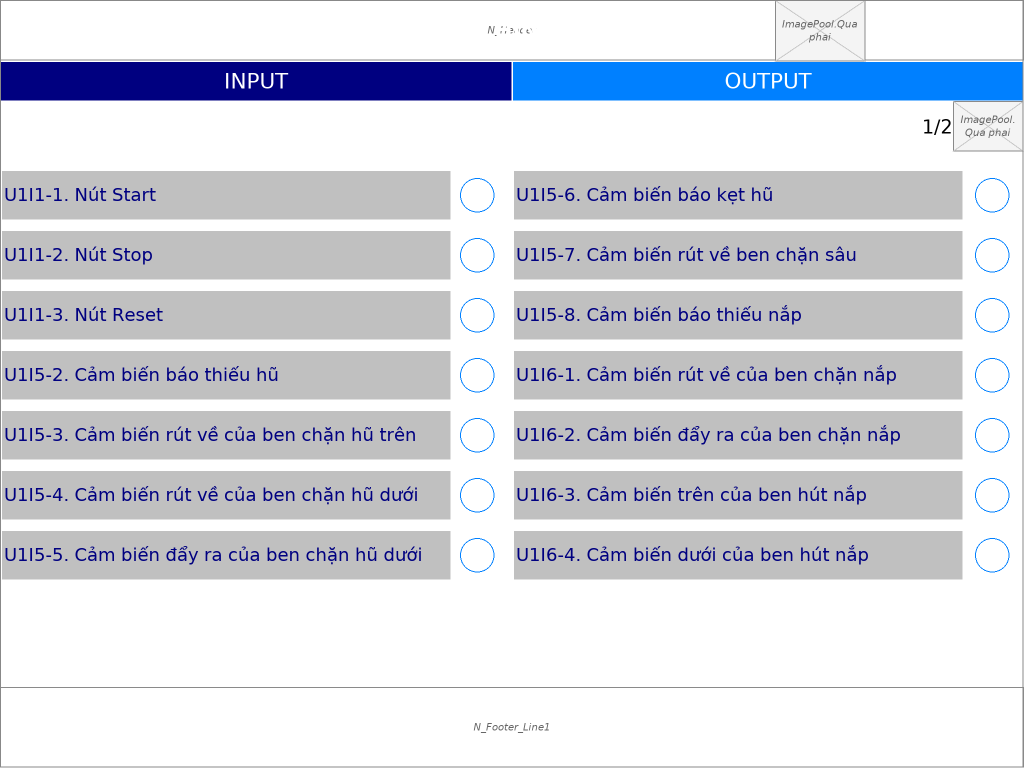
VISUALIZATION N_PLC_I1  // 1024x768
    Frame (0,687 1024x80)
        shows N_Footer_Line1()
    Frame (0,0 1024x60)
        shows N_Header()
    Textfield (353,5 400x50), "MÀN HÌNH IO LINE 1"
    Rectangle (0,61 512x40), "INPUT"
        OnMouseClick: change screen: N_PLC_I1
    Rectangle (512,61 512x40), "OUTPUT"
        OnMouseClick: change screen: N_PLC_O1
    Image (775,0 90x61), image: ImagePool.Qua phai
        OnMouseClick: change screen: N_PLC_I2
    Rectangle (1,350 450x50), "U1I5-2. Cảm biến báo thiếu hũ"
    Rectangle (1,410 450x50), "U1I5-3. Cảm biến rút về của ben chặn hũ trên"
    Rectangle (1,470 450x50), "U1I5-4. Cảm biến rút về của ben chặn hũ dưới"
    Rectangle (1,530 450x50), "U1I5-5. Cảm biến đẩy ra của ben chặn hũ dưới"
    Rectangle (1,170 450x50), "U1I1-1. Nút Start"
    Rectangle (1,230 450x50), "U1I1-2. Nút Stop"
    Rectangle (1,290 450x50), "U1I1-3. Nút Reset"
    Ellipse (460,178 34x34), colour toggle: GVL_IO.bStart, input disabled if: true
    Ellipse (460,238 34x34), colour toggle: GVL_IO.bStop, input disabled if: true
    Ellipse (460,298 34x34), colour toggle: GVL_IO.bReset, input disabled if: true
    Ellipse (460,358 34x34), colour toggle: PR_Line01.fb_CupSupply.bCupEmpty, input disabled if: true
    Ellipse (460,418 34x34), colour toggle: PR_Line01.fb_CupSupply.fbCylinder_Up.bAtRetract, input disabled if: true
    Ellipse (460,478 34x34), colour toggle: PR_Line01.fb_CupSupply.fbCylinder_Dw.bAtRetract, input disabled if: true
    Ellipse (460,538 34x34), colour toggle: PR_Line01.fb_CupSupply.fbCylinder_Dw.bAtExtend, input disabled if: true
    Rectangle (513,530 450x50), "U1I6-4. Cảm biến dưới của ben hút nắp"
    Rectangle (513,170 450x50), "U1I5-6. Cảm biến báo kẹt hũ"
    Rectangle (513,230 450x50), "U1I5-7. Cảm biến rút về ben chặn sâu"
    Rectangle (513,290 450x50), "U1I5-8. Cảm biến báo thiếu nắp"
    Rectangle (513,350 450x50), "U1I6-1. Cảm biến rút về của ben chặn nắp"
    Rectangle (513,410 450x50), "U1I6-2. Cảm biến đẩy ra của ben chặn nắp"
    Rectangle (513,470 450x50), "U1I6-3. Cảm biến trên của ben hút nắp"
    Ellipse (975,178 34x34), colour toggle: PR_Line01.fb_CupSupply.bCupDrop, input disabled if: true
    Ellipse (975,538 34x34), colour toggle: PR_Line01.fb_LidSupply.fbCylinder_Suction.bAtExtend, input disabled if: true
        toggle GVL_OF_VU.bSensorOutOfLid[2]
    Ellipse (975,238 34x34), colour toggle: PR_Line01.fb_WormWeight.fbCylinder.bAtRetract, input disabled if: true
    Ellipse (975,298 34x34), colour toggle: PR_Line01.fb_LidSupply.bLidEmpty, input disabled if: true
    Ellipse (975,358 34x34), colour toggle: PR_Line01.fb_LidSupply.fbCylinder_LidStopper.bAtRetract, input disabled if: true
    Ellipse (975,418 34x34), colour toggle: PR_Line01.fb_LidSupply.fbCylinder_LidStopper.bAtExtend, input disabled if: true
    Ellipse (975,478 34x34), colour toggle: PR_Line01.fb_LidSupply.fbCylinder_Suction.bAtRetract, input disabled if: true
    Rectangle (886,102 103x50), "1/2"
    Image (953,101 70x50), image: ImagePool.Qua phai
        OnMouseClick: change screen: N_PLC_I1_next
END_VISUALIZATION

(* stored: Version 1.1.0.1, ProductVersion 3.1.4024.12
   Visu N_PLC_I1: Id {bab97a24-7ed7-451c-b3bc-f4581a93367a} *)
